FUNCTION F_WriteRawVarint32 : HRESULT
VAR_IN_OUT
    aBuffer : ARRAY [*] OF BYTE;
    stState : ST_WriterInternalState;
END_VAR
VAR_INPUT
    anyVarInt32 : ANY_INT;
END_VAR
VAR
    nValue  : UDINT;
END_VAR


IF anyVarInt32.diSize > SIZEOF(UDINT) THEN
    F_WriteRawVarint32 := stState.eWriterErrorCode := E_WriterErrorCode.InvalidDataType;     
    stState.bError := TRUE;
    RETURN; 
END_IF

// Enough capacity left for theoretical max Varint32?
IF (stState.nBufferPos + SIZEOF(nValue) + 1) > stState.nBufferSize THEN
    F_WriteRawVarint32 := stState.eWriterErrorCode := E_WriterErrorCode.TruncatedMessage;     
    stState.bError := TRUE;
    RETURN; 
END_IF

MEMCPY(destAddr:= ADR(nValue), srcAddr:= anyVarInt32.pValue, n:= TO_UDINT(anyVarInt32.diSize));

// fastpath for a common case of single byte value
IF nValue < 16#80 THEN
    aBuffer[stState.nBufferPos] := TO_BYTE(nValue);
    stState.nBufferPos := stState.nBufferPos + 1;
    F_WriteRawVarint32 := S_OK;
    RETURN;
END_IF

WHILE (stState.nBufferPos < stState.nBufferSize) DO
    IF nValue > 16#7F THEN
        aBuffer[stState.nBufferPos] := TO_BYTE((nValue AND 16#7F) OR 16#80);
        nValue := SHR(nValue, 7);
        stState.nBufferPos := stState.nBufferPos + 1;
    ELSE
        aBuffer[stState.nBufferPos] := TO_BYTE(nValue);
        stState.nBufferPos := stState.nBufferPos + 1;
        F_WriteRawVarint32 := S_OK;
        RETURN;
    END_IF
END_WHILE

// should never reach
F_WriteRawVarint32 := E_WriterErrorCode.InternalError;

END_FUNCTION

(* stored: Version 1.1.0.1
   POU F_WriteRawVarint32: Id {1ebc98d9-6b9e-427e-9469-28c03076e903}, SpecialFunc None *)
